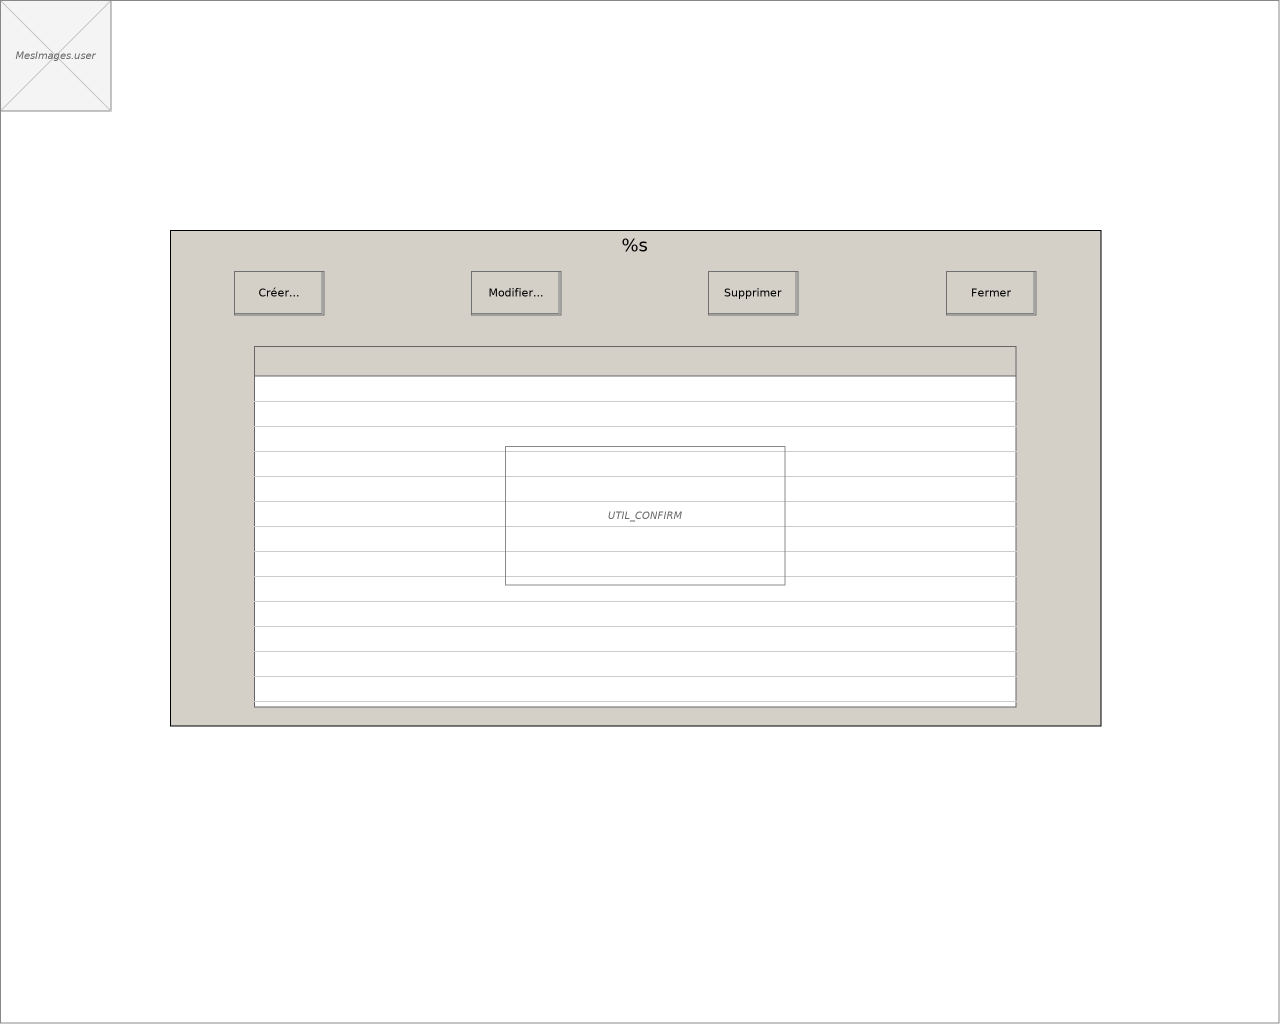
VISUALIZATION UTIL_USER  // 1280x1024
    RoundedRectangle (170,230 931x496)
    Image (0,0 111x111), image: MesImages.user
    Table (254,346 762x361), data array: PRG_USER.TBL_USER
        p1137915858: PRG_USER.LIGNE
        p3854506369: PRG_USER.TBL_USER[INDEX].LOGIN
        p1892666644: PRG_USER.TBL_USER[INDEX].PASS
        p338671338: PRG_USER.TBL_USER[INDEX].PASS_DISPLAY
        p2170511999: PRG_USER.TBL_USER[INDEX].NOM
        p3723444502: PRG_USER.TBL_USER[INDEX].PRENOM
        p1218418051: PRG_USER.TBL_USER[INDEX].GROUPE
        p2232123230: Identifiant
        p4092479075: Nom
        p2237128397: Prenom
        p505689113: Groupe
    Textfield (231,233 808x25), "%s", text list: 'TextList_Util_Userlist', text index: 4
    Button (234,271 90x44), "Créer...", invisible if: PRG_USER.STOP_USER
        toggle PRG_USER.DD_EFFACE_NEW
        OnMouseClick: change screen: UTIL_NEW_USER
    Button (471,271 90x44), "Modifier...", input disabled if: NOT PRG_USER.AUT_MOD_USER
        toggle PRG_USER.DD_mod_user1
        OnMouseClick: change screen: UTIL_MOD_USER
    Button (708,271 90x44), "Supprimer", input disabled if: NOT PRG_USER.AUT_MOD_USER
        toggle PRG_USER.VISU_FEN3
    Button (946,271 90x44), "Fermer", input disabled if: PRG_USER.VISU_FEN3
        OnMouseClick: change screen: UTIL_MENU
    Frame (505,446 280x139), invisible if: NOT PRG_USER.VISU_FEN3
        shows UTIL_CONFIRM(Num_Text := 18, OrdreDD := PRG_USER.DD_DEL_USER, Visu := PRG_USER.VISU_FEN3)
END_VISUALIZATION

(* stored: Version 1.1.0.1, ProductVersion 3.1.4024.10
   Visu UTIL_USER: Id {3a2c1bf6-05ab-43e6-9543-d7375e98191d} *)
